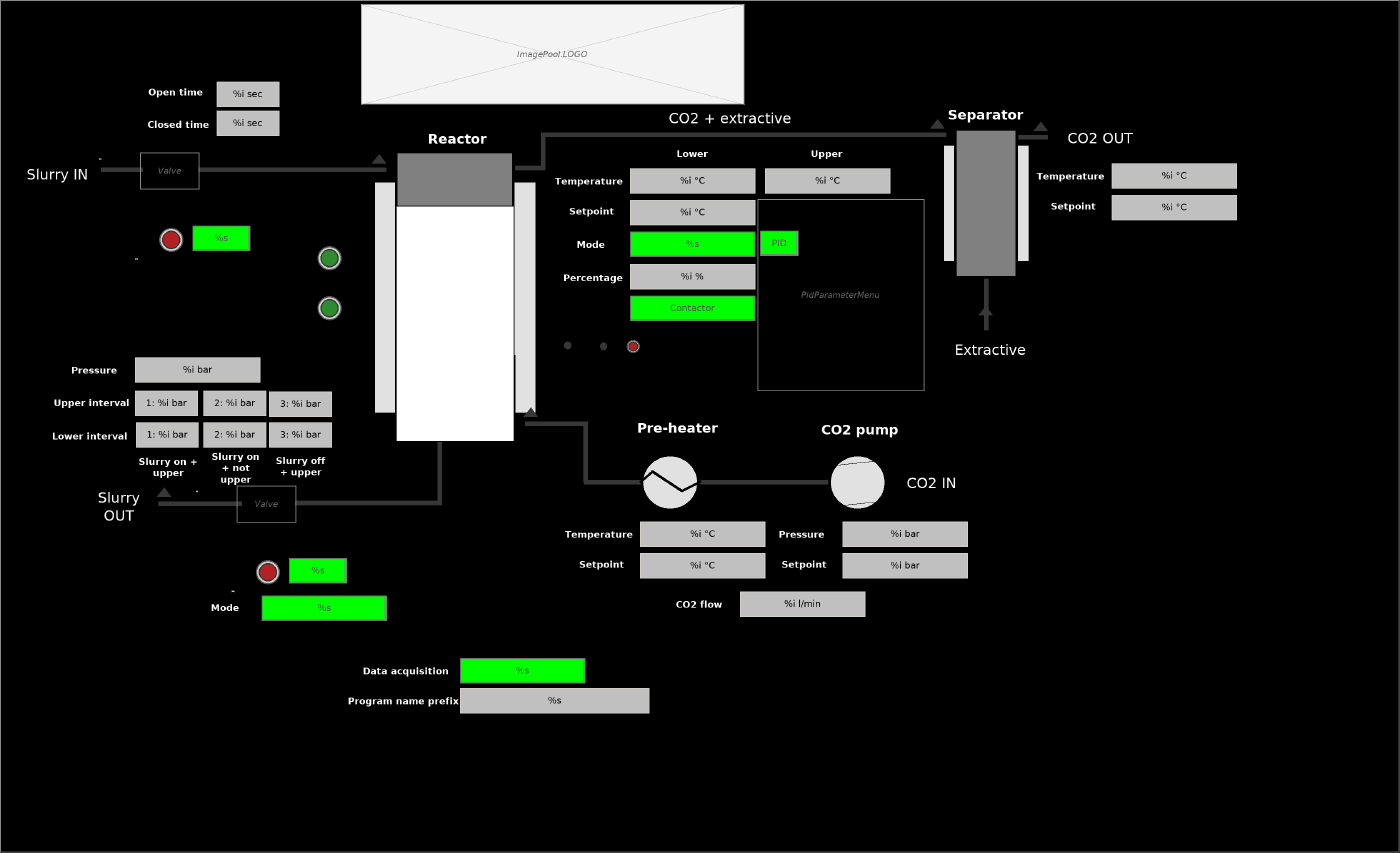
VISUALIZATION MainScreen_1  // 1680x1024
    Line (473,367) (407,367)
    Line (473,308) (407,308)
    Rectangle (1181,326 5x70)
    Rectangle (701,576 350x5)
    Rectangle (525,526 5x80), colour toggle: GVL_IO.reactorOutletValve
    Rectangle (190,602 100x5), colour toggle: GVL_IO.reactorOutletValve
    Rectangle (354,601 175x5), colour toggle: GVL_IO.reactorOutletValve
    Rectangle (121,201 50x5), colour toggle: GVL_IO.reactorInletValve
    Polygon (446,196) (455,185) (463,196) (457,196) (452,196), colour toggle: GVL_IO.reactorInletValve
    Rectangle (238,201 225x5), colour toggle: GVL_IO.reactorInletValve
    Textfield (918,202 150x30), "%i °C", text variable: ReactorTemperatureControl.iTemperatureLowerDisplayValue
    Rectangle (1130,172 107x144)
    Rectangle (447,216 198x282), colour toggle: (ReactorTemperatureControl.bTemperatureControlSwitch) OR (ReactorTemperatureControl.iTemperatureControlPercentage > 0) OR ((ReactorTemperatureControl.iTemperatureControlPercentage = 0) AND (GVL_IO.reactorTemperatureContactor = 1))
    RoundedRectangle (474,181 143x345)
    Button (756,355 150x30), "Contactor", colour toggle: GVL_IO.reactorTemperatureContactor, invisible if: ReactorTemperatureControl.iTemperatureControlPercentage > 0 or ReactorTemperatureControl.bTemperatureControlSwitch= 1
        toggle GVL_IO.reactorTemperatureContactor
    Lamp1 (746,407 28x18), variable: GVL_IO.reactorTemperatureContactor, style: Lamp-Lamp1-Red
    Lamp1 (379,351 33x38), variable: GVL_IO.reactorLevelLow, style: Lamp-Lamp1-Green
    Lamp1 (379,291 33x38), variable: GVL_IO.reactorLevelHigh, style: Lamp-Lamp1-Green
    Textfield (756,240 150x30), "%i °C", text variable: ReactorTemperatureControl.iTemperatureSetpoint
        OnMouseDown: write the text variable via VisuDialogs.Numpad, min 40, max 120
    Label (636,196 142x44), "Temperature"
    Button (756,278 150x30), "%s", text variable: ReactorTemperatureControl.sTemperatureControlState, colour toggle: ReactorTemperatureControl.bTemperatureControlSwitch
        toggle ReactorTemperatureControl.bTemperatureControlSwitch
    Label (638,272 142x44), "Mode"
    Label (639,232 142x44), "Setpoint"
    Textfield (756,202 150x30), "%i °C", text variable: ReactorTemperatureControl.iTemperatureDisplayValue
    RoundedRectangle (474,426 144x101), invisible if: (NOT GVL_IO.reactorLevelLowerLow) OR (GVL_IO.reactorLevelHigh)
    Label (474,152 150x30), "Reactor"
    RoundedRectangle (474,367 143x162), invisible if: (NOT GVL_IO.reactorLevelHigh) OR (GVL_IO.reactorLevelLow)
    RoundedRectangle (474,307 143x223), invisible if: (NOT GVL_IO.reactorLevelLow) OR (GVL_IO.reactorLevelHigherHigh)
    RoundedRectangle (475,247 142x283), invisible if: (NOT GVL_IO.reactorLevelHigherHigh)
    Image (278,709 3x1), image: VisuSymbols.Symbols.TriangleRight
    Line (354,638) (288,638)
    Lamp1 (305,668 33x38), variable: GVL_IO.reactorOutletValve, style: Lamp-Lamp1-Red
    Label (641,312 142x44), "Percentage", invisible if: ReactorTemperatureControl.bTemperatureControlSwitch
    Textfield (756,317 150x30), "%i %", text variable: ReactorTemperatureControl.iTemperatureControlPercentage, invisible if: ReactorTemperatureControl.bTemperatureControlSwitch
        OnMouseDown: write the text variable via VisuDialogs.Numpad, min 0, max 100
    Label (199,708 142x44), "Mode"
    Button (314,715 150x30), "%s", text variable: ReactorLevelAndPressureControl.sLevelControlState, colour toggle: ReactorLevelAndPressureControl.bLevelControlSwitch
        toggle ReactorLevelAndPressureControl.bLevelControlSwitch
    Button (347,670 69x30), "%s", text variable: ReactorLevelAndPressureControl.sLevelValveState, colour toggle: GVL_IO.reactorOutletValve, invisible if: ReactorLevelAndPressureControl.sLevelControlState = 'AUTO'
        toggle GVL_IO.reactorOutletValve
    Image (235,589 2x1), image: VisuSymbols.Symbols.ArrowBoldRight
    Image (433,5 460x120), image: ImagePool.LOGO
    Button (912,277 46x30), "PID", invisible if: ReactorTemperatureControl.bTemperatureControlSwitch
        toggle ReactorTemperatureControl.bPIDcontrolParameterMenu
    Frame (909,239 200x230), invisible if: NOT ReactorTemperatureControl.bPIDcontrolParameterMenu OR ReactorTemperatureControl.bTemperatureControlSwitch
        shows PidParameterMenu()
    Label (42,423 142x44), "Pressure"
    Textfield (162,429 150x30), "%i bar", text variable: ReactorLevelAndPressureControl.iPressureScaledValue
    Button (552,790 150x30), "%s", text variable: RunMATLAB.sMatlabRunningState, pressed state: RunMATLAB.bMatlabBtnState, input disabled if: RunMATLAB.dMatlabBtnColor = 16#FFFFFF00
        p2175578022: RunMATLAB.dMatlabBtnColor
        toggle RunMATLAB.bMatlabBtn
    Image (162,310 3x1), image: VisuSymbols.Symbols.TriangleRight
    Line (238,239) (172,239)
    Lamp1 (189,269 33x38), variable: GVL_IO.reactorInletValve, style: Lamp-Lamp1-Red
    Button (231,271 69x30), "%s", text variable: ReactorLevelAndPressureControl.sFillingValveState, colour toggle: GVL_IO.reactorInletValve, invisible if: ReactorLevelAndPressureControl.sLevelControlState = 'AUTO'
        toggle GVL_IO.reactorInletValve
    Image (119,190 2x1), image: VisuSymbols.Symbols.ArrowBoldRight
    Ellipse (769,545 70x68)
    Polyline (768,579) (783,566) (818,589) (840,578) (838,578)
    Ellipse (994,545 70x68)
    Line (994,559) (1052,553)
    Line (994,608) (1052,602)
    Label (648,620 142x44), "Temperature"
    Textfield (768,664 150x30), "%i °C", text variable: SerialCommunicationHandler.preHeaterTemperatureSetpoint
        OnMouseDown: write SerialCommunicationHandler.preHeaterTemperatureSetSetpoint via VisuDialogs.Numpad, min 0, max 120
    Label (651,656 142x44), "Setpoint"
    Textfield (768,626 150x30), "%i °C", text variable: SerialCommunicationHandler.preHeaterTemperatureMeasurement
    Label (891,620 142x44), "Pressure"
    Textfield (1011,664 150x30), "%i bar", text variable: SerialCommunicationHandler.pumpingPressureSetpoint
        OnMouseDown: write SerialCommunicationHandler.pumpingPressureSetSetpoint via VisuDialogs.Numpad, min 80, max 350
    Label (894,656 142x44), "Setpoint"
    Textfield (1011,626 150x30), "%i bar", text variable: SerialCommunicationHandler.pumpingPressureMeasurement
    Label (1073,565 90x30), "CO2 IN"
    Label (957,501 150x30), "CO2 pump"
    Label (738,499 150x30), "Pre-heater"
    Label (98,574 90x69), "Slurry OUT"
    Label (24,175 90x69), "Slurry IN"
    Label (768,704 142x44), "CO2 flow"
    Textfield (888,710 150x30), "%i l/min", text variable: SerialCommunicationHandler.flowMeasurement
    RoundedRectangle (1145,154 76x180)
    Label (1108,123 150x30), "Separator"
    Label (765,127 222x30), "CO2 + extractive"
    Label (1254,151 133x30), "CO2 OUT"
    Label (1122,405 133x30), "Extractive"
    Label (1214,190 142x44), "Temperature"
    Textfield (1334,234 150x30), "%i °C", text variable: SerialCommunicationHandler.separatorTemperatureSetpoint
        OnMouseDown: write SerialCommunicationHandler.separatorTemperatureSetSetpoint via VisuDialogs.Numpad, min 0, max 100
    Label (1217,226 142x44), "Setpoint"
    Textfield (1334,196 150x30), "%i °C", text variable: SerialCommunicationHandler.separatorTemperatureMeasurement
    Label (416,784 142x44), "Data acquisition"
    Label (60,462 100x44), "Upper interval"
    Label (58,502 100x44), "Lower interval"
    Textfield (162,469 75x30), "1: %i bar", text variable: ReactorLevelAndPressureControl.PressureUpperInterVal_1
        OnMouseDown: write the text variable via VisuDialogs.Numpad, min -100, max 100
    Textfield (244,469 75x30), "2: %i bar", text variable: ReactorLevelAndPressureControl.PressureUpperInterVal_2
        OnMouseDown: write the text variable via VisuDialogs.Numpad, min -100, max 100
    Textfield (163,507 75x30), "1: %i bar", text variable: ReactorLevelAndPressureControl.PressureLowerInterval_1
        OnMouseDown: write the text variable via VisuDialogs.Numpad, min -100, max 100
    Textfield (244,507 75x30), "2: %i bar", text variable: ReactorLevelAndPressureControl.PressureLowerInterval_2
        OnMouseDown: write the text variable via VisuDialogs.Numpad, min -100, max 100
    Label (163,89 100x44), "Open time"
    Label (164,128 100x44), "Closed time"
    Textfield (260,98 75x30), "%i sec", text variable: ReactorLevelAndPressureControl.fillingValveOpenInterval
        OnMouseDown: write the text variable via VisuDialogs.Numpad, min 0, max 100
    Textfield (260,133 75x30), "%i sec", text variable: ReactorLevelAndPressureControl.fillingValveCloseInterval
        OnMouseDown: write the text variable via VisuDialogs.Numpad, min 0, max 200
    Label (760,163 142x44), "Lower"
    Label (921,163 142x44), "Upper"
    Textfield (323,470 75x30), "3: %i bar", text variable: ReactorLevelAndPressureControl.PressureUpperInterVal_3
        OnMouseDown: write the text variable via VisuDialogs.Numpad, min -100, max 100
    Textfield (323,507 75x30), "3: %i bar", text variable: ReactorLevelAndPressureControl.PressureLowerInterval_3
        OnMouseDown: write the text variable via VisuDialogs.Numpad, min -100, max 100
    Label (163,539 78x44), "Slurry on + upper"
    Label (325,538 72x44), "Slurry off + upper"
    Label (247,540 72x44), "Slurry on + not upper"
    Textfield (552,826 227x30), "%s", text variable: GVL_OPC.OPC_ProgramNamePrefix
        OnMouseDown: write the text variable via Edit
    Label (413,820 142x44), "Program name prefix"
    Line (677,415) (644,415)
    Ellipse (676,409 10x11)
    Line (719,415) (686,415), invisible if: NOT GVL_IO.reactorTemperatureContactor
    Ellipse (719,410 10x11)
    Line (725,400) (692,400), invisible if: GVL_IO.reactorTemperatureContactor
    Line (746,415) (728,415)
    Frame (168,183 71x44)
        shows Valve(valve_toggleColor := GVL_IO.reactorInletValve, valve_tapVariable := GVL_IO.reactorInletValve)
    Frame (284,583 71x44)
        shows Valve(valve_toggleColor := GVL_IO.reactorOutletValve, valve_tapVariable := GVL_IO.reactorOutletValve)
    Polygon (188,596) (197,585) (205,596) (199,596) (194,596), colour toggle: GVL_IO.reactorOutletValve
    Polygon (628,500) (637,489) (645,500) (639,500) (634,500)
    Rectangle (630,506 75x5)
    Rectangle (700,507 5x72)
    Rectangle (650,159 485x5)
    Polygon (1116,154) (1125,143) (1133,154) (1127,154) (1122,154)
    Rectangle (649,159 5x45)
    Rectangle (618,199 35x5)
    Polygon (1174,378) (1183,367) (1191,378) (1185,378) (1180,378)
    Rectangle (1222,162 35x5)
    Polygon (1240,157) (1249,146) (1257,157) (1251,157) (1246,157)
END_VISUALIZATION

(* stored: Version 1.1.0.1, ProductVersion 3.1.4024.9
   Visu MainScreen_1: Id {825d6c5d-1db4-4d09-9524-d39611e22440} *)
